Staubli VAL3: ReadMe.pgx

program ReadMe()
begin
  //trDownLead
  //rz 圆弧度
  //ry 圆直径

  //bWeldEnable  是否焊接


end
